{attribute addProperty BoxType "EL3773-0000-0018"}
{attribute addProperty Id "I1_StatusAT %I*I1_Status_E2EFACF1162"}
{attribute addProperty CRC "1350428595"}
{attribute addProperty SizeInBites "16"}
{attribute addProperty SizeInBytes "2"}
TYPE L1_Current_Status_507DE7B3 :
STRUCT
	{attribute addProperty Name "I1_Status"}
	I1_Status AT %I* : I1_Status_E2EFACF1;
END_STRUCT
END_TYPE

(* stored: Version 1.2.0.0, ProductVersion 3.1.4024.9
   DUT L1_Current_Status_507DE7B3: Id {c19a564c-8c5d-4436-b336-95ba5250a852} *)
